// TwinCAT 3 PLC project Servo_Drive
// ProgramVersion: 3.1.4024.0
// libraries:
//   Tc2_Standard, * (Beckhoff Automation GmbH)
//   Tc2_System, * (Beckhoff Automation GmbH)
//   Tc3_Module, * (Beckhoff Automation GmbH)
// project tree:
//   / GlobalTextList.TcGTLO, PlcTask.TcTTO, Visualization Manager.TcVMO (not stored)
//   POUs/ LenzeServoDrive.TcPOU, MAIN.TcPOU, SpeedOutputLinearization.TcPOU
//   VISUs/ Visualization.TcVIS

CONFIGURATION Servo_Drive
    RESOURCE PLC ON TwinCAT3
        TASK PlcTask(INTERVAL := T#10ms, PRIORITY := 20);
        PROGRAM MAIN WITH PlcTask : MAIN;
    END_RESOURCE
END_CONFIGURATION

// ---- POUs/MAIN.TcPOU
PROGRAM MAIN
VAR
END_VAR

LenzeServoDrive();

END_PROGRAM

// ---- POUs/LenzeServoDrive.TcPOU
PROGRAM LenzeServoDrive
VAR
	iSpeedPrg AT %I* : INT; // The actual speed of the motor
	iDancerValue AT %I* : INT; // The position value of the dancer
	bChannel12008 AT %Q* : BOOL; // Digital input channels that enables/disables the safety
	bChannel22008 AT %Q* : BOOL;
	Controlword AT %Q* : BYTE; // Control word of the motor used for switching it on and operating with it
	iSetSpeed AT %Q* : INT; // Activating the speed of the motor
	bButton : BOOL; // Button connected with the HMI that enables the movement of the motor
	rActSpeed : LREAL; // Linearized speed of motor
	fbLinear : SpeedOutputLinearization; // Function for linearization
END_VAR

bChannel12008 := TRUE; //turning the safety off
bChannel22008 := TRUE;

iSetSpeed := 3000; //setting the speed

IF bButton THEN
	Controlword := 9; //if the button is pressed set the motor to OP state
ELSE
	Controlword := 0; //else turn it off (set it to ReadyToBeSwitchedON state
END_IF

fbLinear.iInputSpeed := iSpeedPrg; //linearize the speed
rActSpeed := fbLinear.iOutputSpeed;
fbLinear();

END_PROGRAM

// ---- POUs/SpeedOutputLinearization.TcPOU
FUNCTION_BLOCK SpeedOutputLinearization
VAR_INPUT
	iInputSpeed : INT;
END_VAR
VAR_OUTPUT
	iOutputSpeed : LREAL;
END_VAR
VAR
END_VAR

iOutputSpeed := (3000.0/16384.0)*iInputSpeed;

END_FUNCTION_BLOCK

// ---- GlobalTextList.TcGTLO
TEXTLIST GlobalTextList
  616 = '%f'
  168 = 'Motor Speed: %f'
  41 = 'Motor Switch'
END_TEXTLIST

// ---- VISUs/Visualization.TcVIS
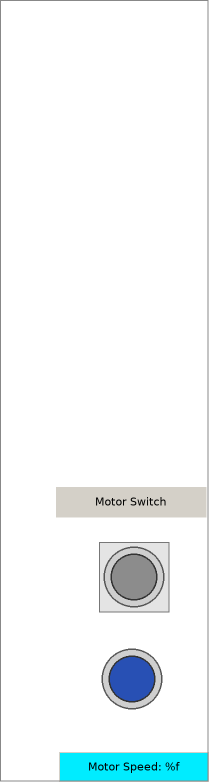
VISUALIZATION Visualization  // 209x782
    Lamp1 (97,644 70x70), variable: LenzeServoDrive.bButton, style: Lamp-Lamp1-Blue
    PushSwitch (99,542 70x70), variable: LenzeServoDrive.bButton, behaviour: TOGGLE, style: Switch-PushSwitch-Gray
    Textfield (56,487 150x30), "Motor Switch", colour toggle: LenzeServoDrive.bButton
    Textfield (59,752 150x30), "Motor Speed: %f", text variable: LenzeServoDrive.rActSpeed
END_VISUALIZATION
